(* Logix 5000 project; controller Generic 1768-L43 rev 15.6; software revision 15.01; part 9 of 10 *)
(* tags used below, declared in another part *)
   Motion_Groups : ALIAS FOR MotionGroup;
   Servo_Axis : ALIAS FOR AXIS_04;
   Servo_CMD : ALIAS FOR Axis_04_CMD;
   Servo_DATA : ALIAS FOR Axis_04_Data;
   Servo_MI : ALIAS FOR Axis_04_MI;
   Servo_STATUS : ALIAS FOR Axis_04_Status;
   Axis_00_CMD : UDT_Axis_CMD;
   Axis_00_Data : UDT_Axis_Data;
   Axis_01_CMD : UDT_Axis_CMD;
   Axis_01_Data : UDT_Axis_Data;
   Axis_01_Status : UDT_Axis_Status;
   Axis_02_CMD : UDT_Axis_CMD;
   Axis_02_Data : UDT_Axis_Data;
   Axis_02_Status : UDT_Axis_Status;
   Axis_03_CMD : UDT_Axis_CMD;
   Axis_03_Data : UDT_Axis_Data;
   Axis_03_Status : UDT_Axis_Status;
   Axis_04_CMD : UDT_Axis_CMD;
   Axis_04_Data : UDT_Axis_Data;
   Axis_04_Status : UDT_Axis_Status;
   ClearFaultDelay : TIMER;
   GenericMachine_COND : UDT_Machine_COND;
   GUI_RunSPD_NI : DINT;
   ManualControl : BOOL;
   PhaseTimout : UDT_PhaseTimeout;
   PZ_GenericMachine_AUTO : PHASE;
(* P05_AXIS_04, continued *)

ROUTINE R01_PowerUP   (* ladder *)
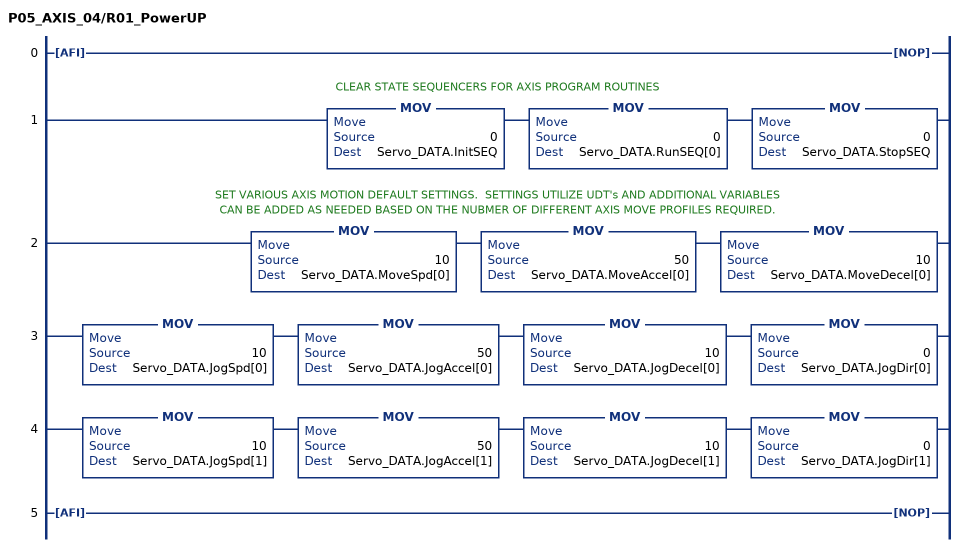
   0: AFI()NOP();
   // CLEAR STATE SEQUENCERS FOR AXIS PROGRAM ROUTINES
   1: MOV(0,Servo_DATA.InitSEQ)MOV(0,Servo_DATA.RunSEQ[0])MOV(0,Servo_DATA.StopSEQ);
   // SET VARIOUS AXIS MOTION DEFAULT SETTINGS.  SETTINGS UTILIZE UDT's AND ADDITIONAL VARIABLES
   // CAN BE ADDED AS NEEDED BASED ON THE NUBMER OF DIFFERENT AXIS MOVE PROFILES REQUIRED.
   2: MOV(10,Servo_DATA.MoveSpd[0])MOV(50,Servo_DATA.MoveAccel[0])MOV(10,Servo_DATA.MoveDecel[0]);
   3: MOV(10,Servo_DATA.JogSpd[0])MOV(50,Servo_DATA.JogAccel[0])MOV(10,Servo_DATA.JogDecel[0])MOV(0,Servo_DATA.JogDir[0]);
   4: MOV(10,Servo_DATA.JogSpd[1])MOV(50,Servo_DATA.JogAccel[1])MOV(10,Servo_DATA.JogDecel[1])MOV(0,Servo_DATA.JogDir[1]);
   5: AFI()NOP();
END_ROUTINE

ROUTINE R02_AxisMonitor   (* ladder *)
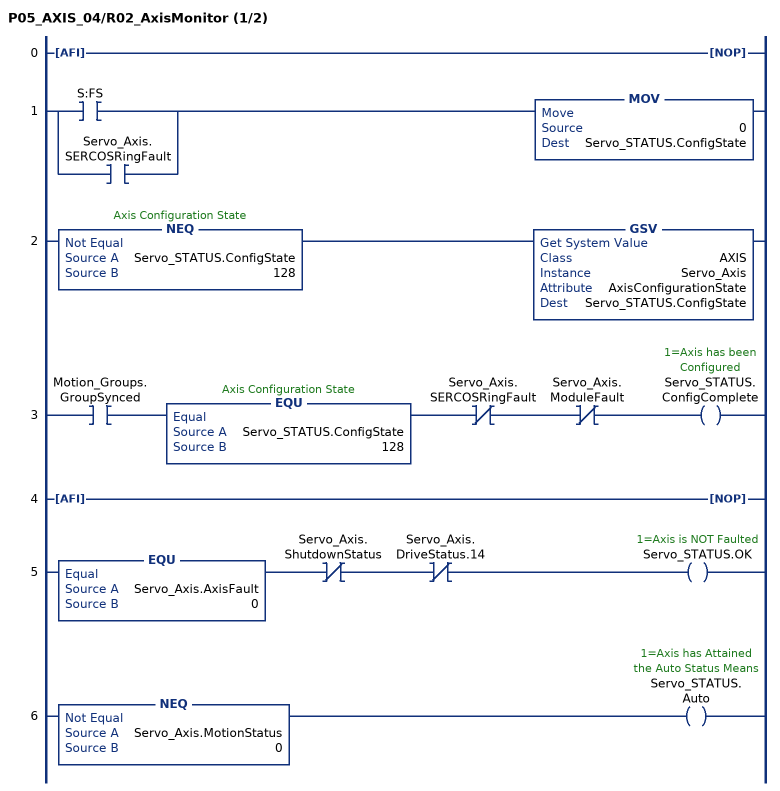
   0: AFI()NOP();
   1: [XIC(S:FS) ,XIC(Servo_Axis.SERCOSRingFault) ]MOV(0,Servo_STATUS.ConfigState);
   2: NEQ(Servo_STATUS.ConfigState,128)GSV(AXIS,Servo_Axis,AxisConfigurationState,Servo_STATUS.ConfigState);
   3: XIC(Motion_Groups.GroupSynced)EQU(Servo_STATUS.ConfigState,128)XIO(Servo_Axis.SERCOSRingFault)XIO(Servo_Axis.ModuleFault)OTE(Servo_STATUS.ConfigComplete);
   4: AFI()NOP();
   5: EQU(Servo_Axis.AxisFault,0)XIO(Servo_Axis.ShutdownStatus)XIO(Servo_Axis.DriveStatus.14)OTE(Servo_STATUS.OK);
   6: NEQ(Servo_Axis.MotionStatus,0)OTE(Servo_STATUS.Auto);
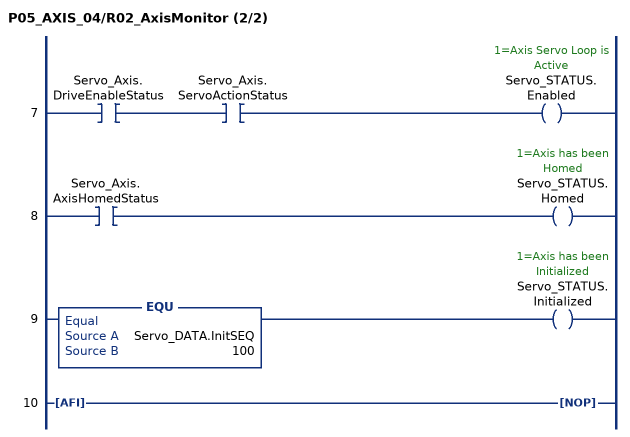
   7: XIC(Servo_Axis.DriveEnableStatus)XIC(Servo_Axis.ServoActionStatus)OTE(Servo_STATUS.Enabled);
   8: XIC(Servo_Axis.AxisHomedStatus)OTE(Servo_STATUS.Homed);
   9: EQU(Servo_DATA.InitSEQ,100)OTE(Servo_STATUS.Initialized);
   10: AFI()NOP();
END_ROUTINE

ROUTINE R03_EnableDisable_FaultReset   (* ladder *)
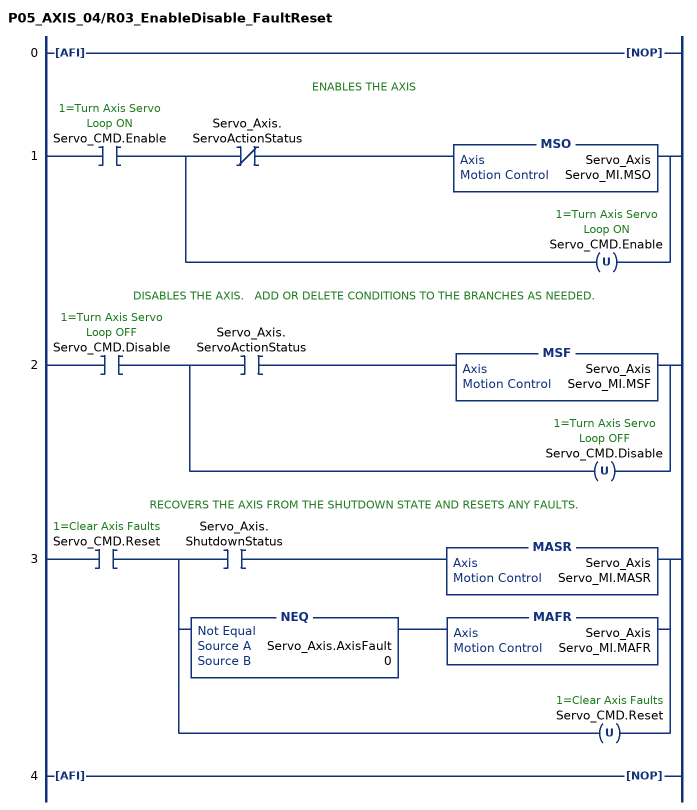
   0: AFI()NOP();
   // ENABLES THE AXIS
   1: XIC(Servo_CMD.Enable)[XIO(Servo_Axis.ServoActionStatus) MSO(Servo_Axis,Servo_MI.MSO) ,OTU(Servo_CMD.Enable) ];
   // DISABLES THE AXIS.   ADD OR DELETE CONDITIONS TO THE BRANCHES AS NEEDED.
   2: XIC(Servo_CMD.Disable)[XIC(Servo_Axis.ServoActionStatus) MSF(Servo_Axis,Servo_MI.MSF) ,OTU(Servo_CMD.Disable) ];
   // RECOVERS THE AXIS FROM THE SHUTDOWN STATE AND RESETS ANY FAULTS.
   3: XIC(Servo_CMD.Reset)[XIC(Servo_Axis.ShutdownStatus) MASR(Servo_Axis,Servo_MI.MASR) ,NEQ(Servo_Axis.AxisFault,0) MAFR(Servo_Axis,Servo_MI.MAFR) ,OTU(Servo_CMD.Reset) ];
   4: AFI()NOP();
END_ROUTINE

ROUTINE R04_Initialize   (* ladder *)
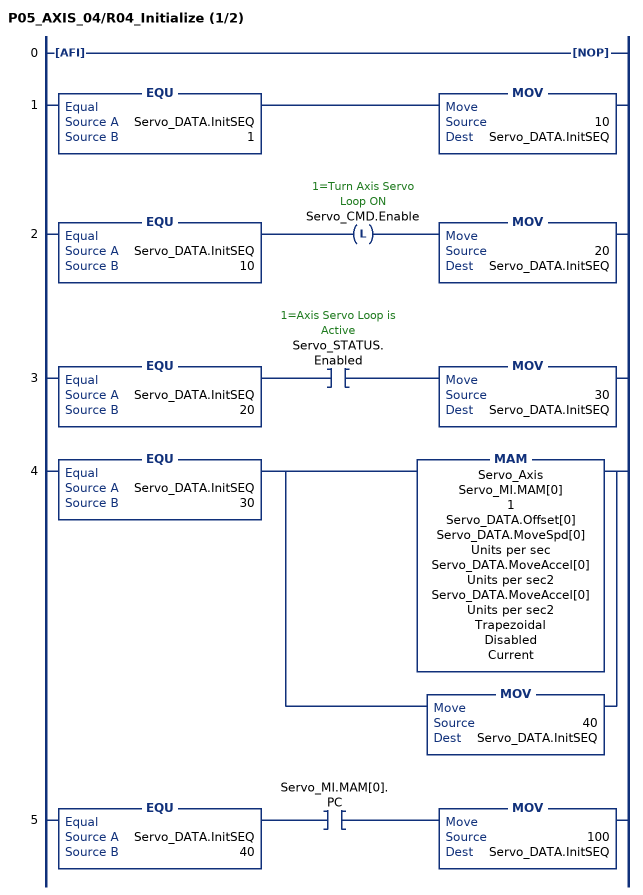
   0: AFI()NOP();
   1: EQU(Servo_DATA.InitSEQ,1)MOV(10,Servo_DATA.InitSEQ);
   2: EQU(Servo_DATA.InitSEQ,10)OTL(Servo_CMD.Enable)MOV(20,Servo_DATA.InitSEQ);
   3: EQU(Servo_DATA.InitSEQ,20)XIC(Servo_STATUS.Enabled)MOV(30,Servo_DATA.InitSEQ);
   4: EQU(Servo_DATA.InitSEQ,30)[MAM(Servo_Axis,Servo_MI.MAM[0],1,Servo_DATA.Offset[0],Servo_DATA.MoveSpd[0],Units per sec,Servo_DATA.MoveAccel[0],Units per sec2,Servo_DATA.MoveAccel[0],Units per sec2,Trapezoidal,Disabled,Current) ,MOV(40,Servo_DATA.InitSEQ) ];
   5: EQU(Servo_DATA.InitSEQ,40)XIC(Servo_MI.MAM[0].PC)MOV(100,Servo_DATA.InitSEQ);
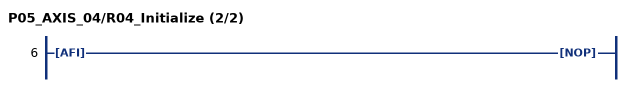
   6: AFI()NOP();
END_ROUTINE

ROUTINE R05_Manual   (* ladder *)
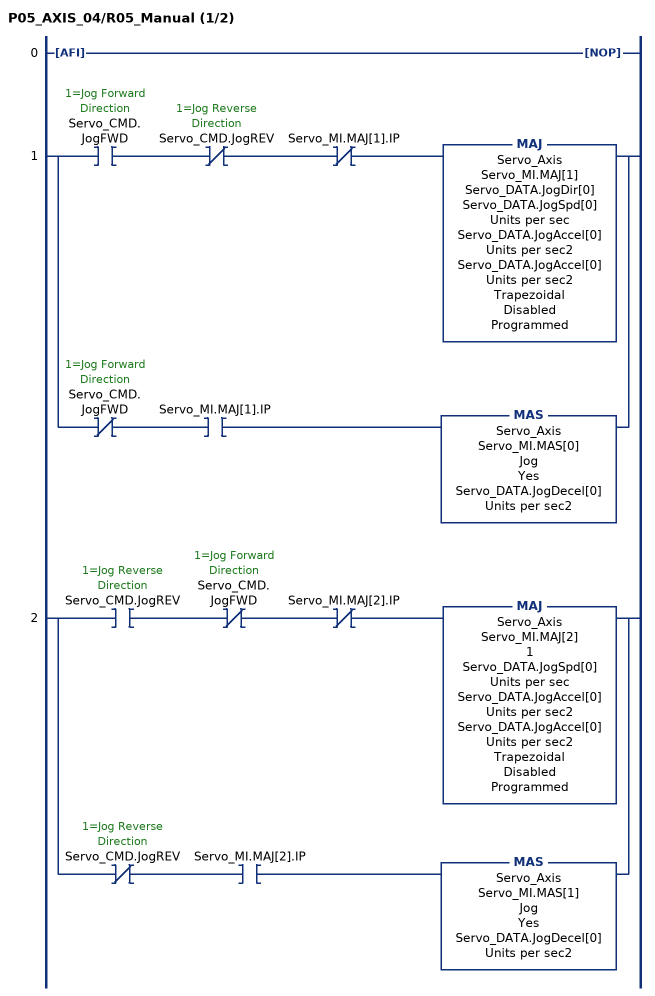
   0: AFI()NOP();
   1: [XIC(Servo_CMD.JogFWD) XIO(Servo_CMD.JogREV) XIO(Servo_MI.MAJ[1].IP) MAJ(Servo_Axis,Servo_MI.MAJ[1],Servo_DATA.JogDir[0],Servo_DATA.JogSpd[0],Units per sec,Servo_DATA.JogAccel[0],Units per sec2,Servo_DATA.JogAccel[0],Units per sec2,Trapezoidal,Disabled,Programmed) ,XIO(Servo_CMD.JogFWD) XIC(Servo_MI.MAJ[1].IP) MAS(Servo_Axis,Servo_MI.MAS[0],Jog,Yes,Servo_DATA.JogDecel[0],Units per sec2) ];
   2: [XIC(Servo_CMD.JogREV) XIO(Servo_CMD.JogFWD) XIO(Servo_MI.MAJ[2].IP) MAJ(Servo_Axis,Servo_MI.MAJ[2],1,Servo_DATA.JogSpd[0],Units per sec,Servo_DATA.JogAccel[0],Units per sec2,Servo_DATA.JogAccel[0],Units per sec2,Trapezoidal,Disabled,Programmed) ,XIO(Servo_CMD.JogREV) XIC(Servo_MI.MAJ[2].IP) MAS(Servo_Axis,Servo_MI.MAS[1],Jog,Yes,Servo_DATA.JogDecel[0],Units per sec2) ];
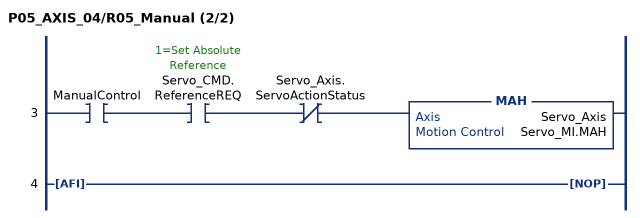
   3: XIC(ManualControl)XIC(Servo_CMD.ReferenceREQ)XIO(Servo_Axis.ServoActionStatus)MAH(Servo_Axis,Servo_MI.MAH);
   4: AFI()NOP();
END_ROUTINE

ROUTINE R06_AutoMotion   (* ladder *)
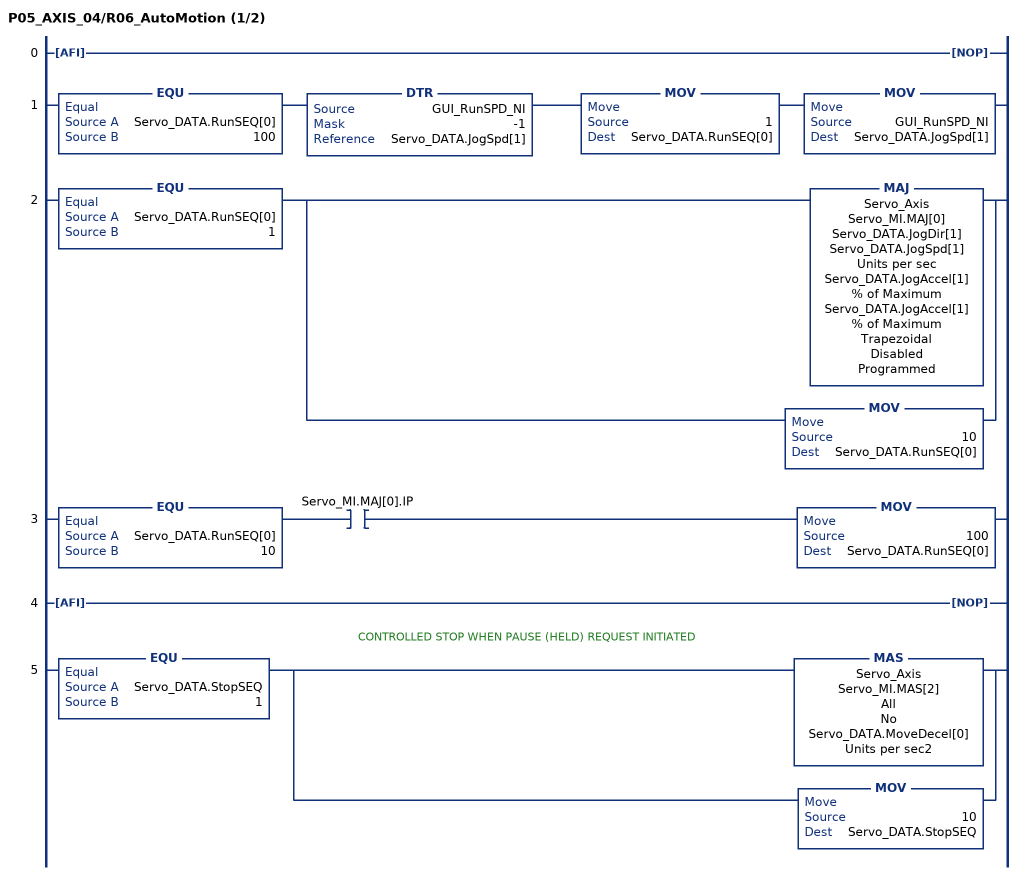
   0: AFI()NOP();
   1: EQU(Servo_DATA.RunSEQ[0],100)DTR(GUI_RunSPD_NI,-1,Servo_DATA.JogSpd[1])MOV(1,Servo_DATA.RunSEQ[0])MOV(GUI_RunSPD_NI,Servo_DATA.JogSpd[1]);
   2: EQU(Servo_DATA.RunSEQ[0],1)[MAJ(Servo_Axis,Servo_MI.MAJ[0],Servo_DATA.JogDir[1],Servo_DATA.JogSpd[1],Units per sec,Servo_DATA.JogAccel[1],% of Maximum,Servo_DATA.JogAccel[1],% of Maximum,Trapezoidal,Disabled,Programmed) ,MOV(10,Servo_DATA.RunSEQ[0]) ];
   3: EQU(Servo_DATA.RunSEQ[0],10)XIC(Servo_MI.MAJ[0].IP)MOV(100,Servo_DATA.RunSEQ[0]);
   4: AFI()NOP();
   // CONTROLLED STOP WHEN PAUSE (HELD) REQUEST INITIATED
   5: EQU(Servo_DATA.StopSEQ,1)[MAS(Servo_Axis,Servo_MI.MAS[2],All,No,Servo_DATA.MoveDecel[0],Units per sec2) ,MOV(10,Servo_DATA.StopSEQ) ];
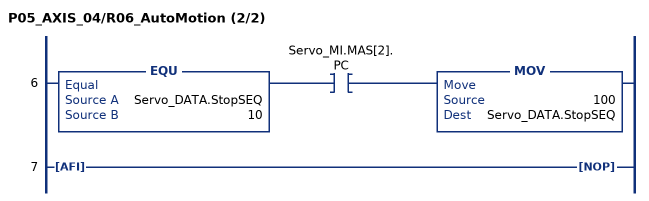
   6: EQU(Servo_DATA.StopSEQ,10)XIC(Servo_MI.MAS[2].PC)MOV(100,Servo_DATA.StopSEQ);
   7: AFI()NOP();
END_ROUTINE
END_PROGRAM

PROGRAM PZ_GenericMachine_AUTO

ROUTINE Aborting   (* ladder *)
// CONTROLS MACHINE ABORTING PHASE.  MODIFY AS NEEDED.
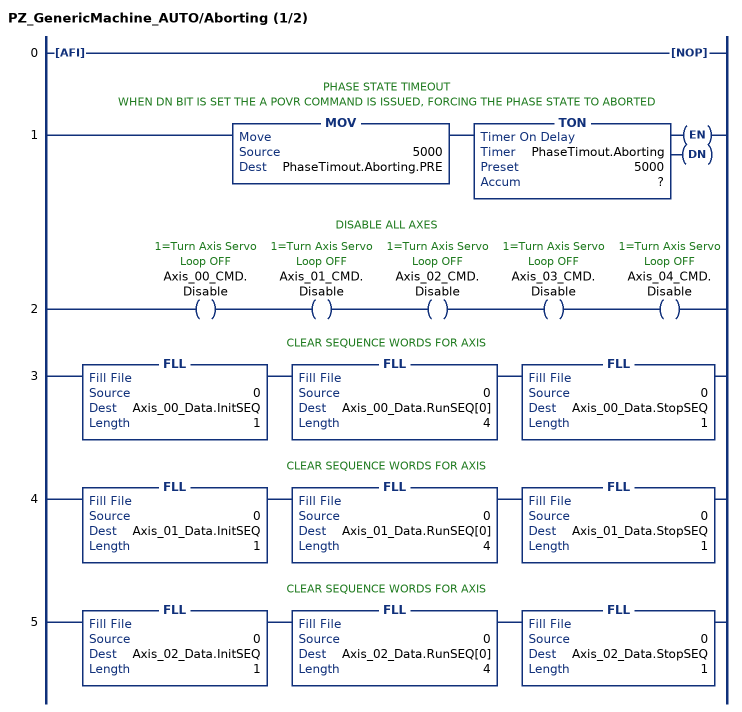
   0: AFI()NOP();
   // PHASE STATE TIMEOUT
   //   WHEN DN BIT IS SET THE A POVR COMMAND IS ISSUED, FORCING THE PHASE STATE TO ABORTED
   1: MOV(5000,PhaseTimout.Aborting.PRE)TON(PhaseTimout.Aborting,?,?);
   // DISABLE ALL AXES
   2: OTE(Axis_00_CMD.Disable)OTE(Axis_01_CMD.Disable)OTE(Axis_02_CMD.Disable)OTE(Axis_03_CMD.Disable)OTE(Axis_04_CMD.Disable);
   // CLEAR SEQUENCE WORDS FOR AXIS
   3: FLL(0,Axis_00_Data.InitSEQ,1)FLL(0,Axis_00_Data.RunSEQ[0],4)FLL(0,Axis_00_Data.StopSEQ,1);
   // CLEAR SEQUENCE WORDS FOR AXIS
   4: FLL(0,Axis_01_Data.InitSEQ,1)FLL(0,Axis_01_Data.RunSEQ[0],4)FLL(0,Axis_01_Data.StopSEQ,1);
   // CLEAR SEQUENCE WORDS FOR AXIS
   5: FLL(0,Axis_02_Data.InitSEQ,1)FLL(0,Axis_02_Data.RunSEQ[0],4)FLL(0,Axis_02_Data.StopSEQ,1);
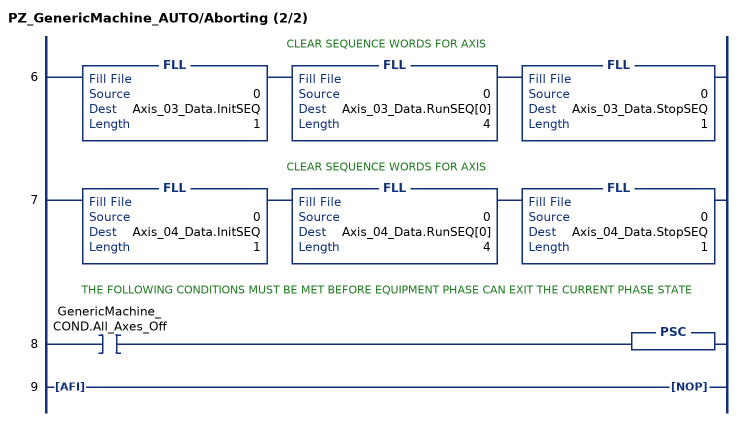
   // CLEAR SEQUENCE WORDS FOR AXIS
   6: FLL(0,Axis_03_Data.InitSEQ,1)FLL(0,Axis_03_Data.RunSEQ[0],4)FLL(0,Axis_03_Data.StopSEQ,1);
   // CLEAR SEQUENCE WORDS FOR AXIS
   7: FLL(0,Axis_04_Data.InitSEQ,1)FLL(0,Axis_04_Data.RunSEQ[0],4)FLL(0,Axis_04_Data.StopSEQ,1);
   // THE FOLLOWING CONDITIONS MUST BE MET BEFORE EQUIPMENT PHASE CAN EXIT THE CURRENT PHASE STATE
   8: XIC(GenericMachine_COND.All_Axes_Off)PSC();
   9: AFI()NOP();
END_ROUTINE

ROUTINE Holding   (* ladder *)
// CONTROLS MACHINE HOLDING PHASE.  MODIFY AS NEEDED.
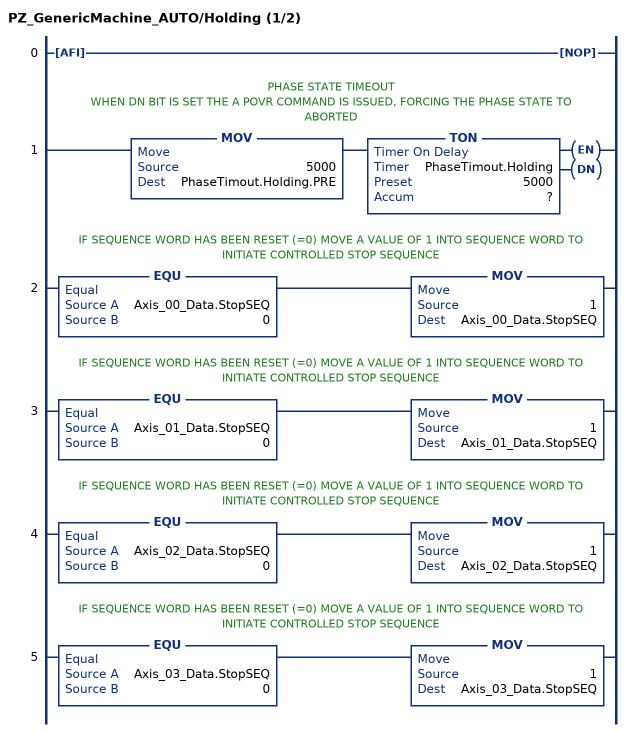
   0: AFI()NOP();
   // PHASE STATE TIMEOUT
   //   WHEN DN BIT IS SET THE A POVR COMMAND IS ISSUED, FORCING THE PHASE STATE TO ABORTED
   1: MOV(5000,PhaseTimout.Holding.PRE)TON(PhaseTimout.Holding,?,?);
   // IF SEQUENCE WORD HAS BEEN RESET (=0) MOVE A VALUE OF 1 INTO SEQUENCE WORD TO INITIATE CONTROLLED STOP SEQUENCE
   2: EQU(Axis_00_Data.StopSEQ,0)MOV(1,Axis_00_Data.StopSEQ);
   // IF SEQUENCE WORD HAS BEEN RESET (=0) MOVE A VALUE OF 1 INTO SEQUENCE WORD TO INITIATE CONTROLLED STOP SEQUENCE
   3: EQU(Axis_01_Data.StopSEQ,0)MOV(1,Axis_01_Data.StopSEQ);
   // IF SEQUENCE WORD HAS BEEN RESET (=0) MOVE A VALUE OF 1 INTO SEQUENCE WORD TO INITIATE CONTROLLED STOP SEQUENCE
   4: EQU(Axis_02_Data.StopSEQ,0)MOV(1,Axis_02_Data.StopSEQ);
   // IF SEQUENCE WORD HAS BEEN RESET (=0) MOVE A VALUE OF 1 INTO SEQUENCE WORD TO INITIATE CONTROLLED STOP SEQUENCE
   5: EQU(Axis_03_Data.StopSEQ,0)MOV(1,Axis_03_Data.StopSEQ);
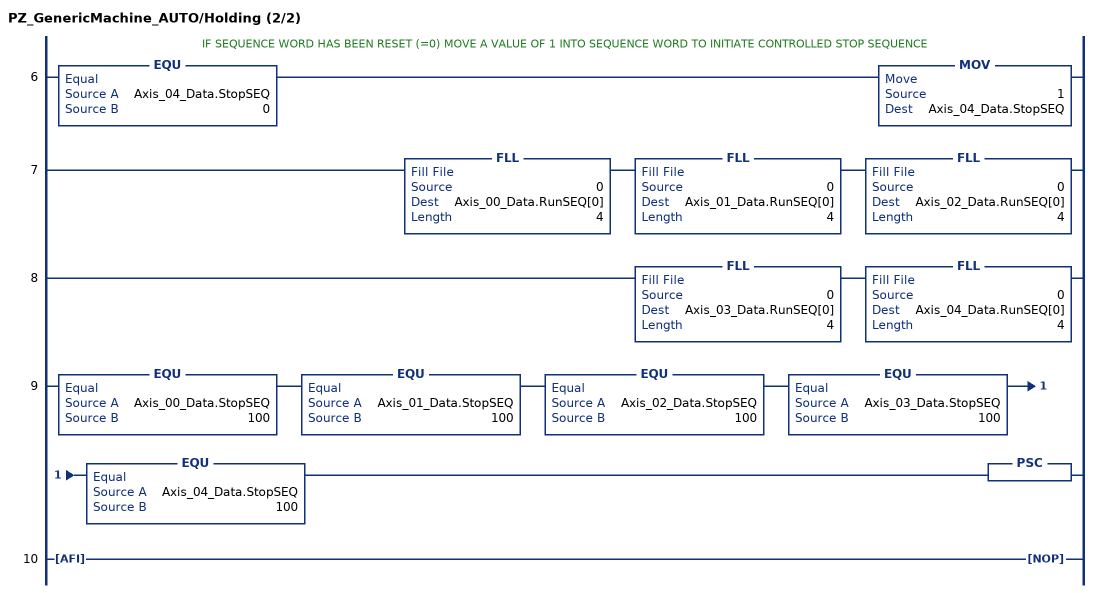
   // IF SEQUENCE WORD HAS BEEN RESET (=0) MOVE A VALUE OF 1 INTO SEQUENCE WORD TO INITIATE CONTROLLED STOP SEQUENCE
   6: EQU(Axis_04_Data.StopSEQ,0)MOV(1,Axis_04_Data.StopSEQ);
   7: FLL(0,Axis_00_Data.RunSEQ[0],4)FLL(0,Axis_01_Data.RunSEQ[0],4)FLL(0,Axis_02_Data.RunSEQ[0],4);
   8: FLL(0,Axis_03_Data.RunSEQ[0],4)FLL(0,Axis_04_Data.RunSEQ[0],4);
   9: EQU(Axis_00_Data.StopSEQ,100)EQU(Axis_01_Data.StopSEQ,100)EQU(Axis_02_Data.StopSEQ,100)EQU(Axis_03_Data.StopSEQ,100)EQU(Axis_04_Data.StopSEQ,100)PSC();
   10: AFI()NOP();
END_ROUTINE

ROUTINE Resetting   (* ladder *)
// CONTROLS MACHINE RESETTING PHASE.  MODIFY AS NEEDED.
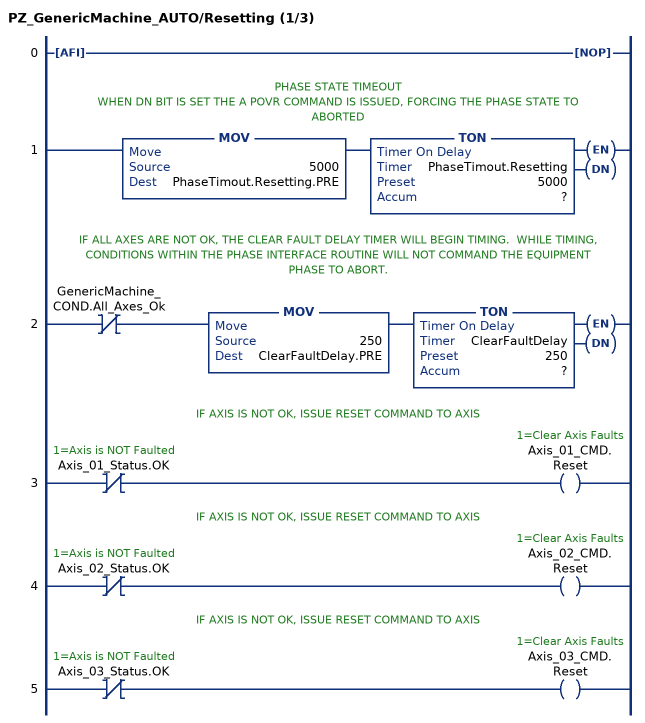
   0: AFI()NOP();
   // PHASE STATE TIMEOUT
   //   WHEN DN BIT IS SET THE A POVR COMMAND IS ISSUED, FORCING THE PHASE STATE TO ABORTED
   1: MOV(5000,PhaseTimout.Resetting.PRE)TON(PhaseTimout.Resetting,?,?);
   // IF ALL AXES ARE NOT OK, THE CLEAR FAULT DELAY TIMER WILL BEGIN TIMING.  WHILE TIMING, CONDITIONS WITHIN THE PHASE INTERFACE ROUTINE WILL NOT COMMAND THE EQUIPMENT PHASE TO ABORT.
   2: XIO(GenericMachine_COND.All_Axes_Ok)MOV(250,ClearFaultDelay.PRE)TON(ClearFaultDelay,?,?);
   // IF AXIS IS NOT OK, ISSUE RESET COMMAND TO AXIS
   3: XIO(Axis_01_Status.OK)OTE(Axis_01_CMD.Reset);
   // IF AXIS IS NOT OK, ISSUE RESET COMMAND TO AXIS
   4: XIO(Axis_02_Status.OK)OTE(Axis_02_CMD.Reset);
   // IF AXIS IS NOT OK, ISSUE RESET COMMAND TO AXIS
   5: XIO(Axis_03_Status.OK)OTE(Axis_03_CMD.Reset);
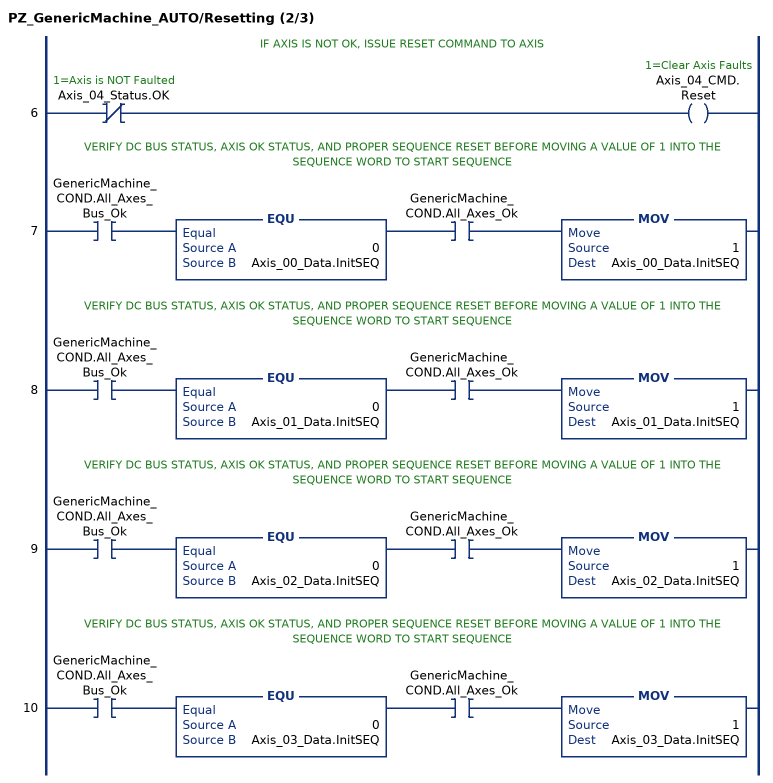
   // IF AXIS IS NOT OK, ISSUE RESET COMMAND TO AXIS
   6: XIO(Axis_04_Status.OK)OTE(Axis_04_CMD.Reset);
   // VERIFY DC BUS STATUS, AXIS OK STATUS, AND PROPER SEQUENCE RESET BEFORE MOVING A VALUE OF 1 INTO THE SEQUENCE WORD TO START SEQUENCE
   7: XIC(GenericMachine_COND.All_Axes_Bus_Ok)EQU(0,Axis_00_Data.InitSEQ)XIC(GenericMachine_COND.All_Axes_Ok)MOV(1,Axis_00_Data.InitSEQ);
   // VERIFY DC BUS STATUS, AXIS OK STATUS, AND PROPER SEQUENCE RESET BEFORE MOVING A VALUE OF 1 INTO THE SEQUENCE WORD TO START SEQUENCE
   8: XIC(GenericMachine_COND.All_Axes_Bus_Ok)EQU(0,Axis_01_Data.InitSEQ)XIC(GenericMachine_COND.All_Axes_Ok)MOV(1,Axis_01_Data.InitSEQ);
   // VERIFY DC BUS STATUS, AXIS OK STATUS, AND PROPER SEQUENCE RESET BEFORE MOVING A VALUE OF 1 INTO THE SEQUENCE WORD TO START SEQUENCE
   9: XIC(GenericMachine_COND.All_Axes_Bus_Ok)EQU(0,Axis_02_Data.InitSEQ)XIC(GenericMachine_COND.All_Axes_Ok)MOV(1,Axis_02_Data.InitSEQ);
   // VERIFY DC BUS STATUS, AXIS OK STATUS, AND PROPER SEQUENCE RESET BEFORE MOVING A VALUE OF 1 INTO THE SEQUENCE WORD TO START SEQUENCE
   10: XIC(GenericMachine_COND.All_Axes_Bus_Ok)EQU(0,Axis_03_Data.InitSEQ)XIC(GenericMachine_COND.All_Axes_Ok)MOV(1,Axis_03_Data.InitSEQ);
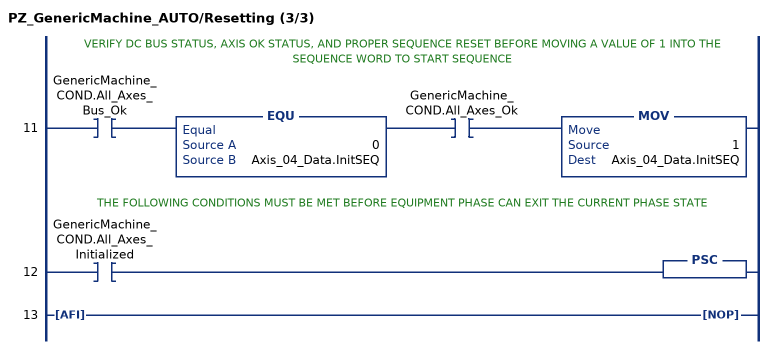
   // VERIFY DC BUS STATUS, AXIS OK STATUS, AND PROPER SEQUENCE RESET BEFORE MOVING A VALUE OF 1 INTO THE SEQUENCE WORD TO START SEQUENCE
   11: XIC(GenericMachine_COND.All_Axes_Bus_Ok)EQU(0,Axis_04_Data.InitSEQ)XIC(GenericMachine_COND.All_Axes_Ok)MOV(1,Axis_04_Data.InitSEQ);
   // THE FOLLOWING CONDITIONS MUST BE MET BEFORE EQUIPMENT PHASE CAN EXIT THE CURRENT PHASE STATE
   12: XIC(GenericMachine_COND.All_Axes_Initialized)PSC();
   13: AFI()NOP();
END_ROUTINE

ROUTINE Restarting   (* ladder *)
// CONTROLS MACHINE RESTARTING PHASE.  MODIFY AS NEEDED.
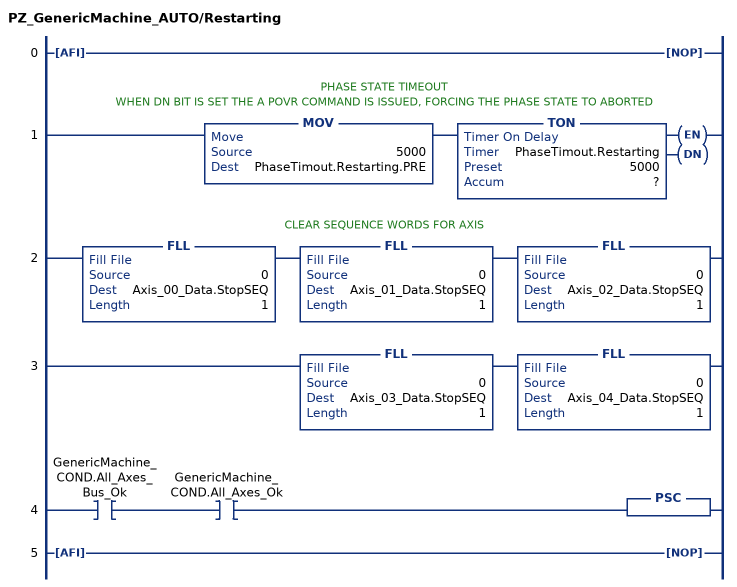
   0: AFI()NOP();
   // PHASE STATE TIMEOUT
   //   WHEN DN BIT IS SET THE A POVR COMMAND IS ISSUED, FORCING THE PHASE STATE TO ABORTED
   1: MOV(5000,PhaseTimout.Restarting.PRE)TON(PhaseTimout.Restarting,?,?);
   // CLEAR SEQUENCE WORDS FOR AXIS
   2: FLL(0,Axis_00_Data.StopSEQ,1)FLL(0,Axis_01_Data.StopSEQ,1)FLL(0,Axis_02_Data.StopSEQ,1);
   3: FLL(0,Axis_03_Data.StopSEQ,1)FLL(0,Axis_04_Data.StopSEQ,1);
   4: XIC(GenericMachine_COND.All_Axes_Bus_Ok)XIC(GenericMachine_COND.All_Axes_Ok)PSC();
   5: AFI()NOP();
END_ROUTINE
